SYSTEM CS21_TEST (* CLIENT_2_1/SERVER_1_2 Test *)
  (* Standard: 61499-1 *)
  (* Version 0.2, 2001-10-12, JHC, Rockwell Automation, Changed CLIENT/SERVER order. *)
  (* Version 0.1, 2001-07-05, JHC, Rockwell Automation, Added TEST application. *)
  (* Version 0.0, 2001-06-02, JHC, Rockwell Automation *)
  APPLICATION TEST
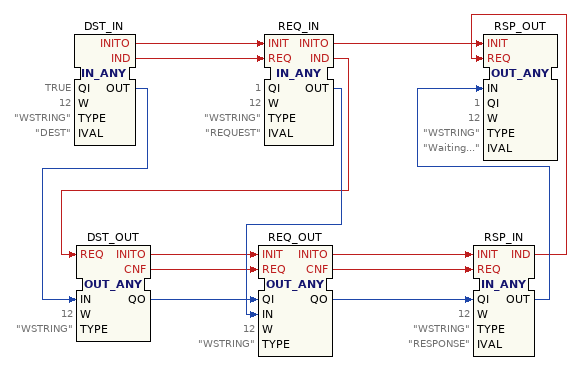
    FBS
      RSP_IN : IN_ANY(W := 12, TYPE := "WSTRING", IVAL := "RESPONSE");
      REQ_OUT : OUT_ANY(W := 12, TYPE := "WSTRING");
      DST_OUT : OUT_ANY(W := 12, TYPE := "WSTRING");
      DST_IN : IN_ANY(QI := TRUE, W := 12, TYPE := "WSTRING", IVAL := "DEST");
      REQ_IN : IN_ANY(QI := 1, W := 12, TYPE := "WSTRING", IVAL := "REQUEST");
      RSP_OUT : OUT_ANY(QI := 1, W := 12, TYPE := "WSTRING", IVAL := "Waiting...");
    END_FBS
    EVENT_CONNECTIONS
      REQ_OUT.INITO TO RSP_IN.INIT;
      REQ_OUT.CNF TO RSP_IN.REQ;
      DST_OUT.INITO TO REQ_OUT.INIT;
      DST_OUT.CNF TO REQ_OUT.REQ;
      DST_IN.INITO TO REQ_IN.INIT;
      DST_IN.IND TO REQ_IN.REQ;
      REQ_IN.INITO TO RSP_OUT.INIT; (* All I/O must be initialized *)
      REQ_IN.IND TO DST_OUT.REQ;
      RSP_IN.IND TO RSP_OUT.REQ;
    END_CONNECTIONS
    DATA_CONNECTIONS
      REQ_OUT.QO TO RSP_IN.QI;
      DST_OUT.QO TO REQ_OUT.QI;
      DST_IN.OUT TO DST_OUT.IN;
      REQ_IN.OUT TO REQ_OUT.IN;
      RSP_IN.OUT TO RSP_OUT.IN;
    END_CONNECTIONS
  END_APPLICATION
  DEVICE CLT : FRAME_DEVICE(BOUNDS := [100,100,125,125], GRID := [1,1])
    RESOURCE RES1 : PANEL_RESOURCE
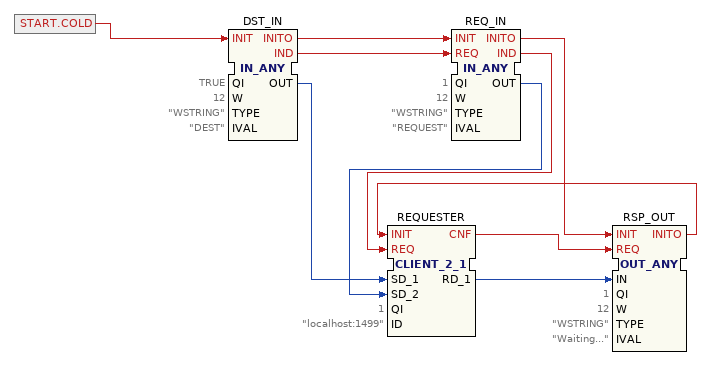
      FBS
        DST_IN : IN_ANY(QI := TRUE, W := 12, TYPE := "WSTRING", IVAL := "DEST");
        REQ_IN : IN_ANY(QI := 1, W := 12, TYPE := "WSTRING", IVAL := "REQUEST");
        REQUESTER : CLIENT_2_1(QI := 1, ID := "localhost:1499");
        RSP_OUT : OUT_ANY(QI := 1, W := 12, TYPE := "WSTRING", IVAL := "Waiting...");
      END_FBS
      EVENT_CONNECTIONS
        START.COLD TO DST_IN.INIT;
        DST_IN.INITO TO REQ_IN.INIT;
        REQ_IN.INITO TO RSP_OUT.INIT; (* All I/O must be initialized *)
        RSP_OUT.INITO TO REQUESTER.INIT; (* before the CLIENT! *)
        DST_IN.IND TO REQ_IN.REQ;
        REQ_IN.IND TO REQUESTER.REQ;
        REQUESTER.CNF TO RSP_OUT.REQ;
      END_CONNECTIONS
      DATA_CONNECTIONS
        DST_IN.OUT TO REQUESTER.SD_1;
        REQ_IN.OUT TO REQUESTER.SD_2;
        REQUESTER.RD_1 TO RSP_OUT.IN;
      END_CONNECTIONS
    END_RESOURCE
  END_DEVICE
  DEVICE SRVR : FRAME_DEVICE(BOUNDS := [225,100,125,125], GRID := [1,1]) (* SERVER must be initialized first! *)
    RESOURCE RES1 : PANEL_RESOURCE
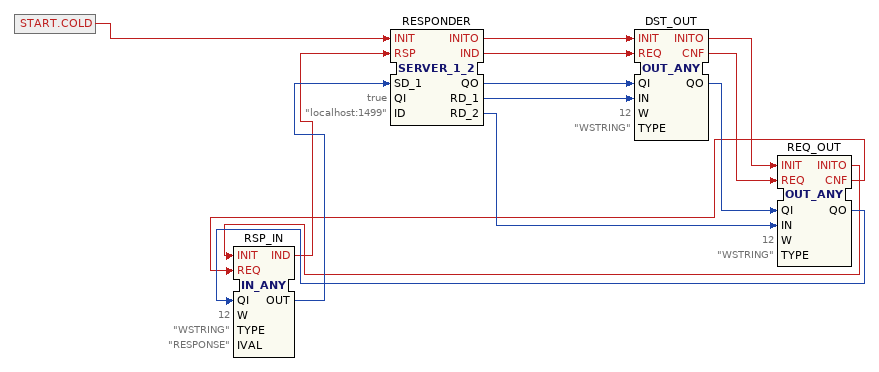
      FBS
        RESPONDER : SERVER_1_2(QI := true, ID := "localhost:1499");
        DST_OUT : OUT_ANY(W := 12, TYPE := "WSTRING");
        REQ_OUT : OUT_ANY(W := 12, TYPE := "WSTRING");
        RSP_IN : IN_ANY(W := 12, TYPE := "WSTRING", IVAL := "RESPONSE");
      END_FBS
      EVENT_CONNECTIONS
        START.COLD TO RESPONDER.INIT;
        RESPONDER.INITO TO DST_OUT.INIT;
        DST_OUT.INITO TO REQ_OUT.INIT;
        REQ_OUT.INITO TO RSP_IN.INIT;
        RESPONDER.IND TO DST_OUT.REQ;
        DST_OUT.CNF TO REQ_OUT.REQ;
        REQ_OUT.CNF TO RSP_IN.REQ;
        RSP_IN.IND TO RESPONDER.RSP;
      END_CONNECTIONS
      DATA_CONNECTIONS
        RESPONDER.QO TO DST_OUT.QI;
        DST_OUT.QO TO REQ_OUT.QI;
        REQ_OUT.QO TO RSP_IN.QI;
        RESPONDER.RD_1 TO DST_OUT.IN;
        RESPONDER.RD_2 TO REQ_OUT.IN;
        RSP_IN.OUT TO RESPONDER.SD_1;
      END_CONNECTIONS
    END_RESOURCE
  END_DEVICE
  MAPPINGS
    TEST.RSP_IN ON RESPONDER.RES1.RSP_IN;
    TEST.REQ_OUT ON RESPONDER.RES1.REQ_OUT;
    TEST.DST_OUT ON RESPONDER.RES1.DST_OUT;
    TEST.DST_IN ON REQUESTER.RES1.DST_IN;
    TEST.REQ_IN ON REQUESTER.RES1.REQ_IN;
    TEST.RSP_OUT ON REQUESTER.RES1.RSP_OUT;
  END_MAPPINGS
END_SYSTEM
